FUNCTION_BLOCK W3W4
  (* Standard: 61499-2 *)
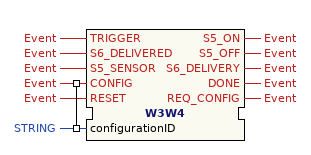
  EVENT_INPUT
    TRIGGER;
    S6_DELIVERED;
    S5_SENSOR;
    CONFIG WITH configurationID;
    RESET;
  END_EVENT
  EVENT_OUTPUT
    S5_ON;
    S5_OFF;
    S6_DELIVERY;
    DONE;
    REQ_CONFIG;
  END_EVENT
  VAR_INPUT
    configurationID : STRING;
  END_VAR
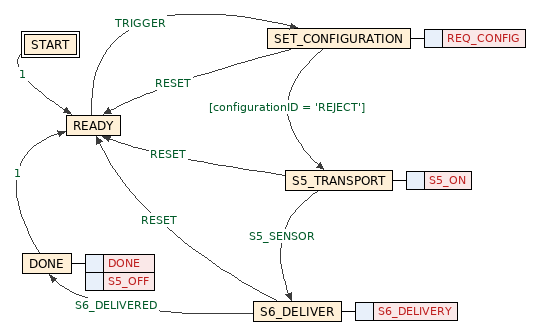
  EC_STATES
    START;
    S5_TRANSPORT : -> S5_ON;
    S6_DELIVER : -> S6_DELIVERY;
    DONE : -> DONE, -> S5_OFF;
    READY;
    SET_CONFIGURATION : -> REQ_CONFIG;
  END_STATES
  EC_TRANSITIONS
    START TO READY := 1;
    S5_TRANSPORT TO S6_DELIVER := S5_SENSOR;
    S6_DELIVER TO DONE := S6_DELIVERED;
    READY TO SET_CONFIGURATION := TRIGGER;
    SET_CONFIGURATION TO S5_TRANSPORT := [configurationID = 'REJECT'];
    DONE TO READY := 1;
    SET_CONFIGURATION TO READY := RESET;
    S5_TRANSPORT TO READY := RESET;
    S6_DELIVER TO READY := RESET;
  END_TRANSITIONS
  ALGORITHM INIT IN ST:

  END_ALGORITHM
  ALGORITHM REQ IN ST:

  END_ALGORITHM
END_FUNCTION_BLOCK
